{attribute 'qualified_only'}
VAR_GLOBAL
	Axis1 : AXIS_REF;
	Axis2 : AXIS_REF;
END_VAR

(* stored: Version 1.1.0.1, ProductVersion 3.1.4024.12
   GVL GVL: Id {a2f49835-1774-4f6e-980c-595da97cc3c9} *)
